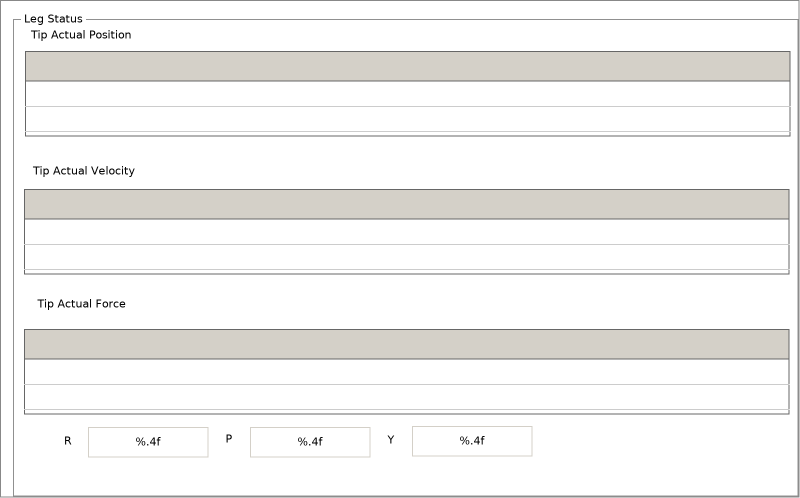
VISUALIZATION Monitor  // 800x498
    GroupBox (13,11 785x485), "Leg Status"
        Table (12,40 765x85), data array: GVL.tipActualPos
            p3854506369: GVL.tipActualPos[0,INDEX]
            p1892666644: GVL.tipActualPos[1,INDEX]
            p338671338: GVL.tipActualPos[2,INDEX]
            p2170511999: GVL.tipActualPos[3,INDEX]
            p3723444502: GVL.tipActualPos[4,INDEX]
            p1218418051: GVL.tipActualPos[5,INDEX]
            p2232123230: LegA
            p511219082: LegB
            p1755163831: LegC
            p4092479075: LegD
            p2237128397: LegE
            p505689113: LegF
        Table (11,178 765x85), data array: GVL.tipActualVel
            p3854506369: GVL.tipActualVel[0,INDEX]
            p1892666644: GVL.tipActualVel[1,INDEX]
            p338671338: GVL.tipActualVel[2,INDEX]
            p2170511999: GVL.tipActualVel[3,INDEX]
            p3723444502: GVL.tipActualVel[4,INDEX]
            p1218418051: GVL.tipActualVel[5,INDEX]
            p2232123230: LegA
            p511219082: LegB
            p1755163831: LegC
            p4092479075: LegD
            p2237128397: LegE
            p505689113: LegF
        Label (16,9 105x30), "Tip Actual Position"
        Label (6,145 130x30), "Tip Actual Velocity"
        Label (20,278 115x30), "Tip Actual Force"
        Table (11,318 765x85), data array: GVL.tipActualFce
            p3854506369: GVL.tipActualFce[0,INDEX]
            p1892666644: GVL.tipActualFce[1,INDEX]
            p338671338: GVL.tipActualFce[2,INDEX]
            p2170511999: GVL.tipActualFce[3,INDEX]
            p3723444502: GVL.tipActualFce[4,INDEX]
            p1218418051: GVL.tipActualFce[5,INDEX]
            p2232123230: LegA
            p511219082: LegB
            p1755163831: LegC
            p4092479075: LegD
            p2237128397: LegE
            p505689113: LegF
        Textfield (75,416 120x30), "%.4f", text variable: GVL.rpy_model[0]
        Textfield (237,416 120x30), "%.4f", text variable: GVL.rpy_model[1]
        Textfield (399,415 120x30), "%.4f", text variable: GVL.rpy_model[2]
        Label (356,414 44x30), "Y"
        Label (194,413 44x30), "P"
        Label (33,415 44x30), "R"
END_VISUALIZATION

(* stored: Version 1.1.0.1, ProductVersion 3.1.4024.2
   Visu Monitor: Id {60bdc1e7-dfbd-41d9-85cc-ddd637a991c7} *)
